Fanuc KAREL source: kt00476.KL

-- PROVISIONAL review KL for V940-1; original PC SHA256 db335ceb763f74a844df119da4418f843ace87931424ed149d5ed4d5990b0cf7
-- Incomplete behavior may be omitted. Consult companion uncertainty JSON. Do not deploy.
PROGRAM KT00476
%NOLOCKGROUP
-- UNRESOLVED_DECL P1 type=000101
-- UNRESOLVED_DECL P2 type=000101
-- UNRESOLVED_DECL OUT type=000106
BEGIN
  -- V9_ZERO_TABLE_METADATA_HINT layout=0001; no indexed target words; source/name/runtime held
  -- UNRESOLVED_PC offsets 5-34; opcodes 49,49,60,7E,4A
  -- UNRESOLVED_PC offsets 39-43; opcodes 7F
END KT00476
